(* IEC 61131-3 sources: AxTestProject/Program/LStandardLibrary, 8 files *)

(* ---- AnalogSignal.st ---- *)
NAMESPACE stdLib.SignalHandling
    CLASS AnalogSignal

        VAR PRIVATE
            m_status : AnalogSignalStatus;
            m_Old : BOOL;
            m_LimiterEnabled : BOOL := FALSE;
            m_minValue : LREAL;
            m_maxValue : LREAL;
        END_VAR

        //##################################################################
        // Method EnableLimiter
        //
        // Enables limitation for analog signal. If limitation enabled,
        // the status bits "MinLimitReached" and "MaxLimitReached" will be
        // set, if the signal exceeds the limits.
        //
        // min : minimal limitation
        // max : max limitation
        //##################################################################
        METHOD PUBLIC EnableLimiter
            VAR_INPUT
                min : LREAL;
                max : LREAL;
            END_VAR
            m_minValue := min;
            m_maxValue := max;
            m_LimiterEnabled := TRUE;
        END_METHOD

        //##################################################################
        // Method DisableLimiter
        //
        // Disables limitation for analog signal. If limitation disabled,
        // the status bits "MinLimitReached" and "MaxLimitReached" will not
        // set, if the signal exceeds the limits.
        //##################################################################
        METHOD PUBLIC DisableLimiter
            m_LimiterEnabled := FALSE;
        END_METHOD

        //##################################################################
        // Method execute
        //
        // Executes the signal evaluation
        //
        //
        //##################################################################
        METHOD PUBLIC execute : AnalogSignalStatus
            VAR_INPUT
                signal : LREAL;
                enable : BOOL := TRUE;
                qDefault : LREAL := 0.0;
                Norm : LREAL := LREAL#1.0;
            END_VAR
            VAR_TEMP
                actValue : LREAL;
            END_VAR
            IF (enable) THEN
                actValue := signal;
                m_status.QBAD := FALSE;
            ELSE
                actValue := qDefault;
                m_status.QBAD := TRUE;
            END_IF;

            // Check Limits if enabled
            IF (m_LimiterEnabled) THEN
                m_status.MaxLimitReached := (actValue >= m_maxValue);
                m_status.MinLimitReached := (actValue <= m_minValue);
            ELSE
                m_status.MaxLimitReached := FALSE;
                m_status.MinLimitReached := FALSE;
            END_IF;

            execute := m_status;

        END_METHOD

    END_CLASS

    TYPE AnalogSignalStatus : STRUCT
            Q : LREAL;
            QBad : BOOL;
            MaxLimitReached : BOOL;
            MinLimitReached : BOOL;
        END_STRUCT;
    END_TYPE

END_NAMESPACE

(* ---- binSignal_copy.st ---- *)
NAMESPACE stdLib.SignalHandling
    CLASS BinSignal

        VAR PRIVATE
            m_status : BinSignalStatus;
            m_Old : BOOL;
        END_VAR

        METHOD PUBLIC execute : BinSignalStatus
            VAR_INPUT
                signal : BOOL;
                enable : BOOL := TRUE;
                qDefault : BOOL := FALSE;
            END_VAR
            VAR_TEMP
                sig : BOOL;
            END_VAR
            IF (enable) THEN
                sig := signal;
                m_status.QBAD := FALSE;
            ELSE
                sig := qDefault;
                m_status.QBAD := TRUE;
            END_IF;

            m_Status.QRis := sig AND NOT(m_Old);
            m_Status.QFal := NOT(sig) AND m_Old;
            m_Old := sig;

            execute := m_status;
        END_METHOD

    END_CLASS

    TYPE BinSignalStatus : STRUCT
            Q : BOOL;
            QRis : BOOL;
            QFal : BOOL;
            QBad : BOOL;
        END_STRUCT;
    END_TYPE

END_NAMESPACE

(* ---- cEncoder.st ---- *)
NAMESPACE stdLib.SignalHandling
    CLASS Encoder
        VAR PRIVATE
            m_aOld : BOOL;
            m_bOld : BOOL;
            m_status : EncoderStatus;
        END_VAR

        // Reset encoder position to zero
        METHOD Reset
            m_status.position := DINT#0;
        END_METHOD

        //Set encoder to specific position
        METHOD Set
            VAR_INPUT
                position : DINT;
            END_VAR
                m_Status.position := position;
                ;
        END_METHOD

        //Evaluate encoder signals A and B
        METHOD PUBLIC evaluate
            VAR_INPUT
                a : BOOL;
                b : BOOL;
            END_VAR
            VAR_TEMP
                aRis : BOOL;
                bRis : BOOL;
                aFal : BOOL;
                bFal : BOOL;
            END_VAR

            aRis := a AND NOT(m_aOld);
            aFal := NOT(a) AND m_aOld;
            m_aOld := a;

            bRis := b AND NOT(m_bOld);
            bFal := NOT(b) AND m_bOld;
            m_bOld := b;

            //Forward detection
            IF (
                aRis AND NOT(b)
                OR a AND bRis
                OR aFal AND b
                OR NOT(a) AND bFal) THEN
                m_status.isInMotion := true;
                m_status.direction := false;
                m_status.position := m_status.position + DINT#1;
                m_status.increments := m_status.increments + DINT#1;
            //Reverse detection
            ELSIF
            (
                aRis AND b
                OR NOT(a) AND bRis
                OR aFal AND NOT(b)
                OR a AND bFal) THEN
                m_status.isInMotion := true;
                m_status.direction := true;
                m_status.position := m_status.position - DINT#1;
                m_status.increments := m_status.increments - DINT#1;
            ELSE
                m_status.isInMotion := false;
                m_status.direction := false;
            END_IF;

        END_METHOD

        METHOD PUBLIC GetStatus : EncoderStatus
            ;
            GetStatus := m_status;
            m_status.increments := DINT#0;
        END_METHOD
    END_CLASS

    TYPE EncoderStatus :
        STRUCT
            position : DINT;  // increments since last reset
            increments : DINT; // increments since last GetStatus-Call
            direction : BOOL; // 0: forward; 1: reverse
            isInMotion : BOOL; // encoder is in motion
        END_STRUCT;
    END_TYPE
END_NAMESPACE

NAMESPACE StdLibTesting
    {Test(a := 1, b := 0, aOld := 0, bOld := 0, dir := 0, pos := DINT#1)}
    {Test(a := 1, b := 1, aOld := 1, bOld := 0, dir := 0, pos := DINT#1)}
    {Test(a := 0, b := 1, aOld := 1, bOld := 1, dir := 0, pos := DINT#1)}
    {Test(a := 0, b := 0, aOld := 0, bOld := 1, dir := 0, pos := DINT#1)}

    {Test(a := 1, b := 1, aOld := 0, bOld := 1, dir := 1, pos := DINT#-1)}
    {Test(a := 0, b := 1, aOld := 0, bOld := 0, dir := 1, pos := DINT#-1)}
    {Test(a := 0, b := 0, aOld := 1, bOld := 0, dir := 1, pos := DINT#-1)}
    {Test(a := 1, b := 0, aOld := 1, bOld := 1, dir := 1, pos := DINT#-1)}

    FUNCTION EncoderDirection
        VAR_INPUT
            a : INT;
            b : INT;
            aOld : INT;
            bOld : INT;
            dir : INT;
            pos : DINT;
        END_VAR
        VAR
            tA : BOOL;
            tB : BOOL;
            tAOld : BOOL;
            tBOld : BOOL;
            tDir : BOOL;
            o : stdLib.SignalHandling.Encoder;
            status : stdLib.SignalHandling.EncoderStatus;
        END_VAR
        tA := a <> 0;
        tB := b <> 0;
        tAOld := aOld <> 0;
        tBold := bOld <> 0;
        tDir := dir <> 0;
        o.Evaluate(tAOld, tBOld);
        o.Evaluate(tA, tB);
        status := o.GetStatus();

        Assert_Equal_BOOL(expected := tDir, actual := status.direction);
        Assert_Equal_DINT(expected := pos, actual := status.position);
        Assert_Equal_DINT(expected := pos, actual := status.increments);

        status := o.GetStatus();
        Assert_Equal_DINT(expected := pos, actual := status.position);
        Assert_Equal_DINT(expected := DINT#0, actual := status.increments);
        ;
    END_FUNCTION
END_NAMESPACE

(* ---- eAxis.st ---- *)
NAMESPACE stdLib
    TYPE
        enStatus : STRUCT
            done : BOOL;
            busy : BOOL;
            error : BOOL;
            status : INT;
        END_STRUCT;
    END_TYPE
END_NAMESPACE

(* ---- tAxisParameter.st ---- *)
NAMESPACE stdLib
    TYPE
        tAxisParameter : STRUCT
            // dynamic values
            maxVelocity : LREAL := 5.0;
            acceleration : LREAL;
            velocity : LREAL;

            // mechanical values
            maxPosition : DINT;
            position : DINT;

        END_STRUCT;
    END_TYPE
END_NAMESPACE

(* ---- tAxisStatus.st ---- *)
NAMESPACE stdLib
    TYPE
        tAxisStatus : STRUCT
            actPosition : DINT;
            isRunning : BOOL;
            hasFault : BOOL;
        END_STRUCT;
    END_TYPE

    //TYPE
    //    arrayOfStruct : ARRAY[0..1] of tAxisStatus := ;
    //END_TYPE

END_NAMESPACE

NAMESPACE Aa
    FUNCTION funcA : Int
        VAR_INPUT
        END_VAR
        VAR_TEMP
        END_VAR
            funcA := 0;
            ;
    END_FUNCTION

    NAMESPACE INTERNAL inner
        FUNCTION innerFunc : Int
            VAR_INPUT
            END_VAR
            VAR_TEMP
            END_VAR

                innerFunc := 1;
        END_FUNCTION
    END_NAMESPACE

    FUNCTION tAxisStatus : Int
        VAR_INPUT
        END_VAR
        VAR_TEMP
            ret : INT;
        END_VAR
        tAxisStatus := inner.innerFunc();

            ;
    END_FUNCTION
END_NAMESPACE

(* ---- Defaults.st ---- *)
NAMESPACE System.Math

    NAMESPACE Const

        FUNCTION PI : LReal
                PI := 3.1415926535897932384626433832795;
        END_FUNCTION

        FUNCTION MaxInt : INT
                MaxInt := 32767;
        END_FUNCTION

        FUNCTION MinInt : INT
                MinInt := -32768;
        END_FUNCTION

        FUNCTION MaxDInt : DINT
                MaxDInt := DINT#32767;
        END_FUNCTION

        FUNCTION MinDInt : DINT
                MinDInt := DINT#-2147483647;
        END_FUNCTION

    END_NAMESPACE

END_NAMESPACE

(* ---- cAxis.st ---- *)
NAMESPACE stdLib
    CLASS Axis

        VAR PUBLIC
            mParameter : tAxisParameter;
            m1 : tAxisParameter;
            mStatus : tAxisStatus;
            run : BOOL;
            faultActive : BOOL;
        END_VAR

        VAR PRIVATE
            mPosition : DINT;
            mAcceleration : LREAL;
            mDeceleration : LREAL;
            mPlcOpenStatus : enStatus;
        END_VAR

        METHOD PUBLIC Main
            ;
        END_METHOD

        METHOD PUBLIC  GetStatus : enStatus
            GetStatus := mPlcOpenStatus;
        END_METHOD

        METHOD PUBLIC  GetInfo : tAxisStatus
            GetInfo := mStatus;
        END_METHOD

        METHOD PUBLIC GetPos : DINT
            GetPos := mPosition;
        END_METHOD

        //--------------------------------------
        // Homing
        //--------------------------------------
        METHOD PUBLIC Homing : enStatus
            VAR_INPUT
                //velocity : LREAL;
                //acceleration : LREAL;
                //deceleration : LREAL;
                //mode : INT;
            END_VAR
            VAR_TEMP
                tempStatus : enStatus;
            END_VAR
                Homing := tempStatus;
        END_METHOD

        METHOD PRIVATE mHoming
            ;
        END_METHOD

        //---------------------------------------------------
        // Reset
        //---------------------------------------------------
        METHOD Reset : BOOL
            VAR_INPUT
            END_VAR
            VAR_TEMP
            END_VAR

            Reset := true;
                ;
        END_METHOD

        //---------------------------------------------------
        // Halt
        //---------------------------------------------------
        METHOD Halt : BOOL
            VAR_INPUT
            END_VAR
            VAR_TEMP
            END_VAR

            Halt := true;
                ;
        END_METHOD

        //---------------------------------------------------
        // MoveVelocity
        //---------------------------------------------------
        METHOD PUBLIC MoveVelocity : BOOL
            VAR_INPUT
                velocity : LREAL;
                acceleration : LREAL;
                deceleration : LREAL;
            END_VAR

            if (not(faultActive)) then
                mPlcOpenstatus.busy := true;
                MoveVelocity := true;
            ELSE
                mPlcOpenstatus.error := true;
                mPlcOpenstatus.busy := false;
                MoveVelocity := false;
            END_IF;

        END_METHOD

        //---------------------------------------------------
        // MoveAbsolute
        //---------------------------------------------------
        METHOD PUBLIC MoveAbsolute : BOOL
            VAR_INPUT
                velocity : LREAL;
                position : DINT;
                acceleration : LREAL;
                deceleration : LREAL;
            END_VAR
            MoveAbsolute := true;
        END_METHOD

        METHOD PUBLIC MoveAbsolute3 : BOOL
            VAR_INPUT
                velocity : LREAL;
                position : DINT;
                acceleration : LREAL;
                deceleration : LREAL;
            END_VAR
            MoveAbsolute3 := true;
        END_METHOD

        //---------------------------------------------------
        // MoveRelative
        //---------------------------------------------------
        METHOD PUBLIC MoveRelative : BOOL
            VAR_INPUT
                velocity : LREAL;
                position : DINT;
                acceleration : LREAL;
                deceleration : LREAL;
            END_VAR
            MoveRelative := true;
        END_METHOD

        //---------------------------------------------------
        // SetAcceleration
        //---------------------------------------------------
        METHOD PUBLIC SetAcceleration
            VAR_INPUT
                accelleration : LREAL;
            END_VAR
            mAcceleration := accelleration;
        END_METHOD

        //---------------------------------------------------
        // SetDeceleration
        //---------------------------------------------------
        METHOD PUBLIC SetDeceleration
            VAR_INPUT
                deceleration : LREAL;
            END_VAR
            mDeceleration := deceleration;
        END_METHOD

        METHOD init
            VAR_INPUT
                parameter : tAxisParameter;
            END_VAR
            ;
            parameter.velocity := 0.0;
            parameter.position := DINT#0;
        END_METHOD

    END_CLASS
END_NAMESPACE
